VISUALIZATION Engineer_HMI  // 1024x768
END_VISUALIZATION

(* stored: Version 1.1.0.1
   Visu Engineer_HMI: Id {3c046ea6-2ad7-430d-94b1-38b7ccc8e80e} *)
